FUNCTION_BLOCK PLCnextMaster (* Service Interface Function Block Type *)
  (* Standard: 61499-2; Description: Copyright (c) 2022 Peirlberger Juergen This program and the accompanying materials are made available under the terms of the Eclipse Public License 2.0 which is available at https://www.eclipse.org/legal/epl-2.0/ SPDX-License-Identifier: EPL-2.0 *)
  (* Version 3.0, 2025-04-14, Patrick Aigner, changed package *)
  (* Version 1.0, 2022-04-07, Peirlberger Juergen *)
  PACKAGE eclipse4diac::io::plcnext;
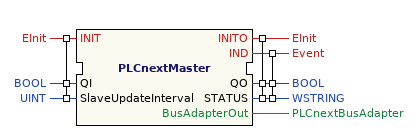
  EVENT_INPUT
    INIT : EInit WITH QI, SlaveUpdateInterval; (* Service Initialization *)
  END_EVENT
  EVENT_OUTPUT
    INITO : EInit WITH QO, STATUS; (* Initialization Confirm *)
    IND WITH QO, STATUS; (* Indication from Resource *)
  END_EVENT
  VAR_INPUT
    QI : BOOL; (* Event Input Qualifier *)
    SlaveUpdateInterval : UINT := 25;
  END_VAR
  VAR_OUTPUT
    QO : BOOL; (* Event Output Qualifier *)
    STATUS : WSTRING; (* Status *)
  END_VAR
  PLUGS
    BusAdapterOut : eclipse4diac::io::plcnext::PLCnextBusAdapter;
  END_PLUGS
END_FUNCTION_BLOCK
